TYPE "Prod_Part_Target"
VERSION : 0.1
// Block: Prod_Part_Target
   STRUCT
      Ready : Bool;
      Tick_Mark : Bool;
      Trace_Mark : Bool;
      P_ID : DInt;
      O_ID : DInt;
      Part_ToGo : DInt;
      Part_Len : Real;
      Part_Tol : Real;
      Beam_Code : Int;
   END_STRUCT;

END_TYPE
